INTERFACE I_Device

METHOD Init : BOOL
VAR_INPUT
    nId : UDINT;
END_VAR
END_METHOD

METHOD Reset
END_METHOD

END_INTERFACE

(* stored: Version 1.1.0.1, ProductVersion 3.1.4024.12
   Itf I_Device: Id {a1b2c3d4-0040-4000-8000-000000000040}
   Method Init: Id {a1b2c3d4-0041-4000-8000-000000000041}
   Method Reset: Id {a1b2c3d4-0042-4000-8000-000000000042} *)
